// TIA Portal V19 export
TYPE "LAF_typeGlobalRuntime"
TITLE = Structure runtime information / Struktur Runtime Informationen
// Type to store the cycle time of the PLC, with maximum, minimum and average values. / Globale Informationen
// stored: Access Published
   STRUCT
      prevCycle : UInt;   // Letzte Zykluszeit / Previous cycle time
      reset : Bool := TRUE;   // Reset Max. / Min. Zykluszeit / Reset max / min cycle time
      maxCycle : UInt;   // Maximale Zykluszeit / Maximum cycle time
      minCycle : UInt := 9999;   // Minimale Zykluszeit / Minimum cycle time
      maxCycleRuntime : UInt;   // Grenzwert Maximale-Zykluszeit / Limit max. cycle time
      minCycleRuntime : UInt;   // Grenzwert Mindest-Zykluszeit / Limit min.cycle time
      maxCommRuntime : Int;   // Grenzwert Kommunikationslast / Limit max. communication load
   END_STRUCT;
END_TYPE
